// Mitsubishi GX Works2 project: 부등호로 카운트   PLC: Q02/Q02H

PROGRAM MAIN
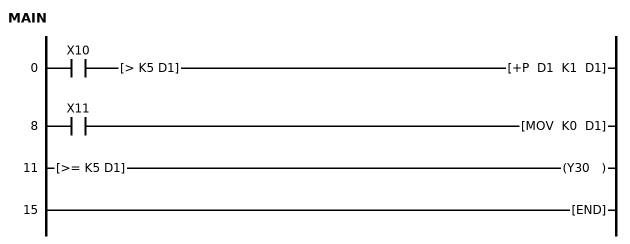
0     LD      X10
      AND>    K5 D1
      +P      D1 K1 D1
8     LD      X11
      MOV     K0 D1
11    LD>=    K5 D1
      OUT     Y30
15    END
END_PROGRAM
